{attribute 'qualified_only'}
VAR_GLOBAL
	PulseOutput		:S_PulseOutput;
	state			:S_State;
END_VAR

(* stored: Version 1.1.0.1, ProductVersion 3.1.4022.16
   GVL GVL_General: Id {9e2d1f25-3e4d-4883-885c-408b2d8ae1b0} *)
